VAR_GLOBAL
	FaultCheck_G : BOOL ; // Test if Fault 
	Fault_Count_G: CTU  ; // Counter 	
	

END_VAR

(* stored: Version 1.1.0.1, ProductVersion 3.1.4024.6
   GVL GVL_Check: Id {1f0ada45-d99d-4ee3-a1db-4792eb1f1fde} *)
